PROGRAM MAIN
VAR
	_Count			: UINT;
END_VAR

_Count := _Count + 1;

END_PROGRAM

(* stored: Version 1.1.0.1
   POU MAIN: Id {aa83fbb2-453b-43e9-a059-eebdb971d1ee}, SpecialFunc None *)
